// TIA Portal V20 export
TYPE "TypeMixerIO"
// stored: IsFailsafeCompliant false
   STRUCT
      Run : Bool;   // Run command in - written by the sequencer each scan, read by the output map.
      SpeedSetpoint { S7_SetPoint := 'True'} : Real := 5.0;   // HMI-tunable - operator units (RPM); the block converts to drive units itself.
      StatusWord : Word;
   END_STRUCT;
END_TYPE
